{attribute 'qualified_only'}
VAR_GLOBAL
	fbTestsuites:			FB_Testsuites;	
END_VAR

(* stored: Version 1.1.0.1
   GVL TestSuiteGVL: Id {cfebde9e-5caa-491e-9955-0f85762b2ab7} *)
